INTERFACE I_StreamReader

{attribute 'monitoring' := 'call'}
PROPERTY BufferAddress : PVOID
GET
END_GET
END_PROPERTY

METHOD GetNextArgTypeId : E_ArgTypeId
END_METHOD

METHOD Read_BLOB
VAR_INPUT
    BlobToCopyTo : ANY;
END_VAR
END_METHOD

METHOD Read_BOOL : BOOL
END_METHOD

METHOD Read_BYTE : BYTE
END_METHOD

METHOD Read_DATA
VAR_INPUT
    DataAddress : PVOID;
    DataLength  : UDINT;
END_VAR
END_METHOD

METHOD Read_DINT : DINT
END_METHOD

METHOD Read_INT : INT
END_METHOD

METHOD Read_LINT : LINT
END_METHOD

METHOD Read_LREAL : LREAL
END_METHOD

METHOD Read_PVOID : PVOID
END_METHOD

METHOD Read_REAL : REAL
END_METHOD

METHOD Read_STRING : STRING(255)
END_METHOD

METHOD Read_STRUCT
VAR_INPUT
    StructureAddress : PVOID;
    StructureLength  : UDINT;
END_VAR
END_METHOD

METHOD Read_UDINT : UDINT
END_METHOD

METHOD Read_UINT : UINT
END_METHOD

METHOD Read_ULINT : ULINT
END_METHOD

{attribute 'monitoring' := 'call'}
PROPERTY ReadPosition : UDINT
GET
END_GET
END_PROPERTY

METHOD SetReadPosition : I_StreamWriter
VAR_INPUT
    Position : UDINT;
END_VAR
END_METHOD

{attribute 'monitoring' := 'call'}
PROPERTY StreamLength : UDINT
GET
END_GET
END_PROPERTY

{attribute 'monitoring' := 'call'}
PROPERTY WritePosition : UDINT
GET
END_GET
END_PROPERTY

END_INTERFACE

(* stored: Version 1.1.0.1, ProductVersion 3.1.4024.12
   Itf I_StreamReader: Id {4ce154d4-15b3-0d46-1c83-b5e5fa9c119b}
   Folder Methods: Id {b8877614-48d5-0eca-2865-22e970702037}
   Folder Properties: Id {75130885-22fc-4e0d-8fe3-aa4a7e663cab}
   Property BufferAddress: Id {3e7e868f-b25b-48a0-84e8-000cff6224e5}
   Get Get: Id {69958d4a-07ec-44dc-8ac2-ba3d959dc291}
   Method GetNextArgTypeId: Id {d474657b-4850-42c6-984b-cda140e1ca70}
   Method Read_BLOB: Id {f8c9a894-7e28-4c4d-9d66-adf775a9e61a}
   Method Read_BOOL: Id {e1bdd036-7870-0f43-0e36-b5bb859b7000}
   Method Read_BYTE: Id {3ccda0cd-8655-0f56-2bc9-c58e6daa3ce8}
   Method Read_DATA: Id {5700a353-f13b-4fdd-b815-4fd238999da2}
   Method Read_DINT: Id {48ce2b84-3168-03ca-12f0-71cd392d8654}
   Method Read_INT: Id {0148bb1b-7254-009d-3f2a-34f63964ce35}
   Method Read_LINT: Id {6c195aa8-b80e-02db-1b75-c81ae8eff187}
   Method Read_LREAL: Id {759500c4-a674-0ff0-2e2d-d445694ce533}
   Method Read_PVOID: Id {3ebc800b-5c5f-0c00-00d9-41734ef2561d}
   Method Read_REAL: Id {76140bff-57d3-00c0-2b2c-0e5854607f62}
   Method Read_STRING: Id {b6f5d3cd-32d2-0aa1-36c6-26f76c20da1d}
   Method Read_STRUCT: Id {d547bbc2-a9a7-40a2-a606-c957f749b757}
   Method Read_UDINT: Id {bc95bb0c-f0ce-0a03-227c-c8ac3d307b3a}
   Method Read_UINT: Id {cda1de9e-731f-09c7-37ed-3632355d115f}
   Method Read_ULINT: Id {c0f7078d-b578-031e-227a-d5f3c9e4196b}
   Property ReadPosition: Id {275e5991-b379-4755-b185-9bf1434e8de7}
   Get Get: Id {263ef926-da42-4324-8471-28495fe924f3}
   Method SetReadPosition: Id {86b70d1c-7207-094c-05c9-c562e8f29569}
   Property StreamLength: Id {0e34a290-63d6-42a0-bec5-b486da5d7878}
   Get Get: Id {9d317ad7-96de-4f4e-91f8-258145f3db73}
   Property WritePosition: Id {c6296339-9b4d-4d8a-9062-ffe48a0ec171}
   Get Get: Id {362d56c1-c398-44a7-92f9-ccc4ae3f4aa6} *)
